TYPE ST_GantryXYZ_HMI :
    STRUCT
        Config  : ST_GantryXYZ_Config;
		Status 	: ST_GantryXYZ_Status;
		Command 	: ST_GantryXYZ_Command;
		Limits  : ST_GantryXYZ_Limits;
    END_STRUCT
END_TYPE

(* stored: Version 1.1.0.1, ProductVersion 3.1.4024.15
   DUT ST_GantryXYZ_HMI: Id {42282f17-118a-4ed6-b5d0-a5b4c6e076c6} *)
